# EPICS alarm handler configuration: mps_database/bare/alarms/areas/mpln_sps_mp04.alhConfig
GROUP NULL MPLN:SPS:MP04:1
$ALIAS MPS Link Node 194
$GUIDANCE
LTUH MPS
   Group Name: MPLN:SPS:MP04:1
   Summary PV:  MPLN:SPS:MP04:1:STATSUMY
$END
CHANNEL  MPLN:SPS:MP04:1    MPLN:SPS:MP04:1:MPS_EN_RBV		-----
CHANNEL  MPLN:SPS:MP04:1    MPLN:SPS:MP04:1:LC1_MODE_RBV		-----
